SUBAPPLICATION Outputs (* Subapplication Type *)
  (* Standard: 61499-2 *)
  (* Version 1.0, 2023-07-15, franz *)
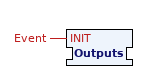
  EVENT_INPUT
    INIT;
  END_EVENT
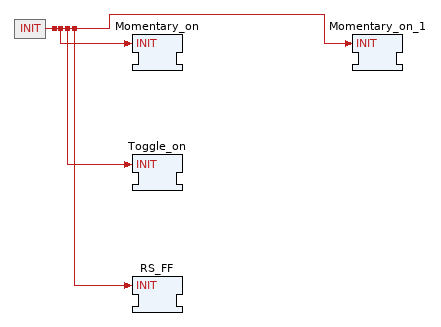
  SUBAPPLICATION Momentary_on (* Tastend Softkey 5000 auf Q1 *)
    EVENT_INPUT
      INIT;
    END_EVENT
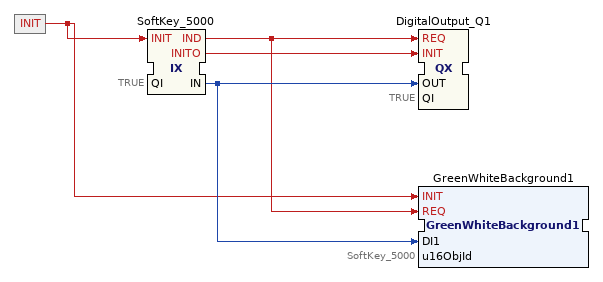
    FBS
      SoftKey_5000 : IX(QI := TRUE);
      DigitalOutput_Q1 : QX(QI := TRUE);
    END_FBS
    SUBAPPS
      GreenWhiteBackground1 : GreenWhiteBackground1(u16ObjId := SoftKey_5000);
    END_SUBAPPS
    EVENT_CONNECTIONS
      SoftKey_5000.IND TO DigitalOutput_Q1.REQ;
      INIT TO SoftKey_5000.INIT;
      INIT TO GreenWhiteBackground1.INIT;
      SoftKey_5000.IND TO GreenWhiteBackground1.REQ;
      SoftKey_5000.INITO TO DigitalOutput_Q1.INIT;
    END_CONNECTIONS
    DATA_CONNECTIONS
      SoftKey_5000.IN TO DigitalOutput_Q1.OUT;
      SoftKey_5000.IN TO GreenWhiteBackground1.DI1;
    END_CONNECTIONS
  END_SUBAPPLICATION
  SUBAPPLICATION Toggle_on (* T-Flip-Flop Softkey 5001 auf Q2 *)
    EVENT_INPUT
      INIT;
    END_EVENT
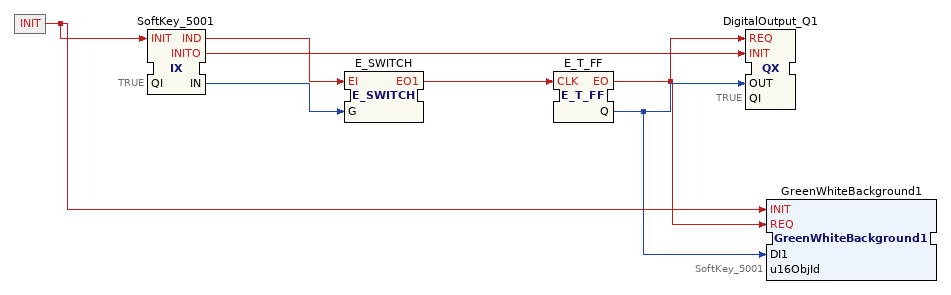
    FBS
      SoftKey_5001 : IX(QI := TRUE);
      DigitalOutput_Q1 : QX(QI := TRUE);
      E_SWITCH : E_SWITCH;
      E_T_FF : E_T_FF;
    END_FBS
    SUBAPPS
      GreenWhiteBackground1 : GreenWhiteBackground1(u16ObjId := SoftKey_5001);
    END_SUBAPPS
    EVENT_CONNECTIONS
      INIT TO SoftKey_5001.INIT;
      INIT TO GreenWhiteBackground1.INIT;
      SoftKey_5001.IND TO E_SWITCH.EI;
      E_SWITCH.EO1 TO E_T_FF.CLK;
      E_T_FF.EO TO DigitalOutput_Q1.REQ;
      SoftKey_5001.INITO TO DigitalOutput_Q1.INIT;
      E_T_FF.EO TO GreenWhiteBackground1.REQ;
    END_CONNECTIONS
    DATA_CONNECTIONS
      SoftKey_5001.IN TO E_SWITCH.G;
      E_T_FF.Q TO DigitalOutput_Q1.OUT;
      E_T_FF.Q TO GreenWhiteBackground1.DI1;
    END_CONNECTIONS
  END_SUBAPPLICATION
  SUBAPPLICATION RS_FF (* T-Flip-Flop Softkey 5002/3 auf Q3 *)
    EVENT_INPUT
      INIT;
    END_EVENT
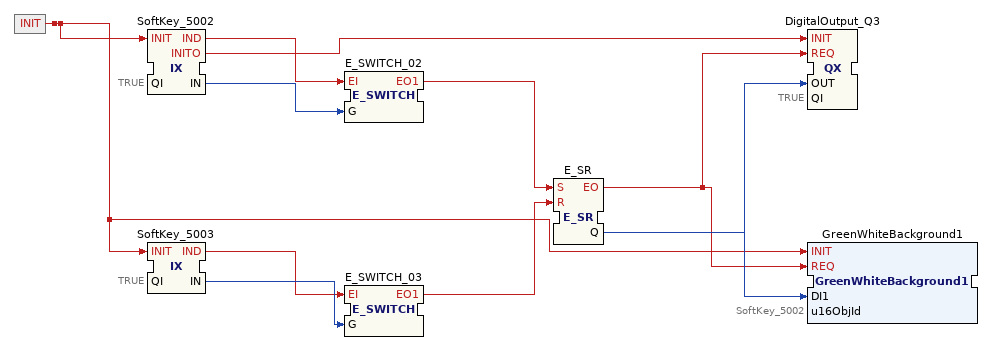
    FBS
      SoftKey_5002 : IX(QI := TRUE);
      DigitalOutput_Q3 : QX(QI := TRUE);
      E_SWITCH_02 : E_SWITCH;
      SoftKey_5003 : IX(QI := TRUE);
      E_SWITCH_03 : E_SWITCH;
      E_SR : E_SR;
    END_FBS
    SUBAPPS
      GreenWhiteBackground1 : GreenWhiteBackground1(u16ObjId := SoftKey_5002);
    END_SUBAPPS
    EVENT_CONNECTIONS
      INIT TO SoftKey_5002.INIT;
      INIT TO GreenWhiteBackground1.INIT;
      SoftKey_5002.IND TO E_SWITCH_02.EI;
      SoftKey_5002.INITO TO DigitalOutput_Q3.INIT;
      SoftKey_5003.IND TO E_SWITCH_03.EI;
      E_SWITCH_02.EO1 TO E_SR.S;
      E_SWITCH_03.EO1 TO E_SR.R;
      E_SR.EO TO DigitalOutput_Q3.REQ;
      E_SR.EO TO GreenWhiteBackground1.REQ;
      INIT TO SoftKey_5003.INIT;
    END_CONNECTIONS
    DATA_CONNECTIONS
      SoftKey_5002.IN TO E_SWITCH_02.G;
      SoftKey_5003.IN TO E_SWITCH_03.G;
      E_SR.Q TO DigitalOutput_Q3.OUT;
      E_SR.Q TO GreenWhiteBackground1.DI1;
    END_CONNECTIONS
  END_SUBAPPLICATION
  SUBAPPLICATION Momentary_on_1 (* Tastend Softkey 5004 und I1 auf Q1 (OR Verknüpfung) *)
    EVENT_INPUT
      INIT;
    END_EVENT
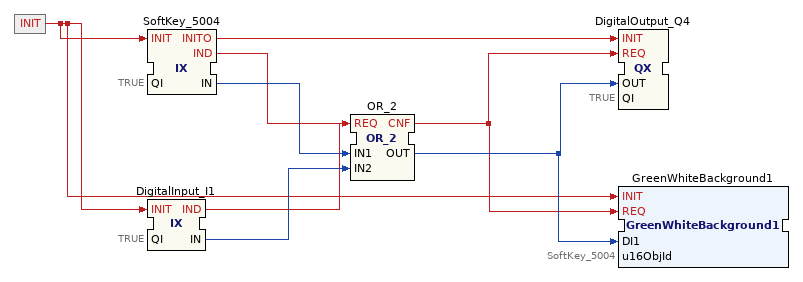
    FBS
      SoftKey_5004 : IX(QI := TRUE);
      DigitalOutput_Q4 : QX(QI := TRUE);
      DigitalInput_I1 : IX(QI := TRUE);
      OR_2 : OR_2;
    END_FBS
    SUBAPPS
      GreenWhiteBackground1 : GreenWhiteBackground1(u16ObjId := SoftKey_5004);
    END_SUBAPPS
    EVENT_CONNECTIONS
      INIT TO SoftKey_5004.INIT;
      INIT TO GreenWhiteBackground1.INIT;
      SoftKey_5004.INITO TO DigitalOutput_Q4.INIT;
      INIT TO DigitalInput_I1.INIT;
      SoftKey_5004.IND TO OR_2.REQ;
      DigitalInput_I1.IND TO OR_2.REQ;
      OR_2.CNF TO DigitalOutput_Q4.REQ;
      OR_2.CNF TO GreenWhiteBackground1.REQ;
    END_CONNECTIONS
    DATA_CONNECTIONS
      SoftKey_5004.IN TO OR_2.IN1;
      DigitalInput_I1.IN TO OR_2.IN2;
      OR_2.OUT TO DigitalOutput_Q4.OUT;
      OR_2.OUT TO GreenWhiteBackground1.DI1;
    END_CONNECTIONS
  END_SUBAPPLICATION
  EVENT_CONNECTIONS
    INIT TO Momentary_on.INIT;
    INIT TO Toggle_on.INIT;
    INIT TO RS_FF.INIT;
    INIT TO Momentary_on_1.INIT;
  END_CONNECTIONS
END_SUBAPPLICATION
